TYPE ST_MotionlinxAI_Axis_HMI :
	STRUCT
		Config	: ST_MotionlinxAI_Axis_Config;
		Command : ST_MotionlinxAI_Axis_Command;
		Status	: ST_MotionlinxAI_Axis_Status;
	END_STRUCT
END_TYPE

(* stored: Version 1.1.0.1, ProductVersion 3.1.4024.15
   DUT ST_MotionlinxAI_Axis_HMI: Id {a8233c30-e0e2-4ae0-9c6e-d86f44760d47} *)
